DATA_BLOCK "DB_Rcv_FIFO_HandOver"
TITLE =%version: 0.11 % CN: 20
//History:
//This version  %created_by:  nltsil %
//              %date_created:  Friday, June 16, 2017 2:11:31 PM %
//              %release: VI_GEN/RA_Dev %
//
//Modification History:                                   By:    Date:     Rev:
//----------------------------------------------------  -------  --------  -----
//ina#5591: Updated Record_Data_Length to 158           nltsil   16-06-17   0.11
//ina#3773: Wrong header, Record_Data_Length to 156     nlHdL    23-01-17   0.10
//ra#9751: Add source files ECS-P to VI_RAW             nlHdL    14-12-15   0.09
//ra#9751: Add source files ECS-P to VI_RAW             nlHdL    07-12-15   0.09
//8673: Reset:Restart for errors via  PNPN interface    nlHdL    29-10-15   0.09
//7324: ECS-P General from the RD to RA for platform    nlHdL    06-07-15   0.08
//23824: Changed Record length to 150                   nlMlaut  29-04-15   0.08
//20643: DB moved to NON RETAIN memory                  nlHdL    16-09-14   0.07
//20899: remove filler from PNPN Lifesign               nlHdL    16-09-14   0.06
//18228: Changed Prefull setting to 16                  nlHHop   28-02-14   0.05
//14210: Header init of FIFO DB                         nlHdL    26-09-13   0.04
//14210: Header init of FIFO DB                         nlHdL    26-09-13   0.03
//15797: Keyword release added                          nlwwij   26-09-13   0.02
//Initial Revision                                      nlHHop   17-04-13   0.01
//
FAMILY : General
VERSION : 0.0
NON_RETAIN


  STRUCT
   General : "UDT_FIFO_PNPN";
   Message : ARRAY  [0 .. 20 ] OF "UDT_PN_Msg_Handover";
  END_STRUCT ;
BEGIN
   General.Status.Empty := TRUE;
   General.Status.Prefull := FALSE;
   General.Status.Full := FALSE;
   General.Status.Record_Length_Too_Long := FALSE;
   General.Status.Wrong_Record_Length := FALSE;
   General.Status.Pointer_Out_Of_Range := FALSE;
   General.Status.Wrong_Prefull_Value := FALSE;
   General.Status.Blockmove_Fault := FALSE;
   General.Status.i_Restart_Request := FALSE;
   General.Status.i_Spare_Request := FALSE;
   General.Status.o_LifeSign_Msgs_Error := FALSE;
   General.Status.o_Spare_Report := FALSE;
   General.Setting.Prefull_Num_Of_Records := 16;
   General.Setting.Record_Data_Length := 158;
   General.Num_Of_Records_stored := 0;
   General.Max_Numb_Of_Records := 0;
   General.Next_Record_store := 0;
   General.Next_Record_Retrieve := 0;
END_DATA_BLOCK

